% RSLogix 500 project I2P JOB 13 B - Andrew.RSS, saved by version 10.00.00.00 %
PROJECT "ML05B"    % processor: Bul.1763 MicroLogix 1100 Series B %

PROGRAM FILES
  LAD 2   13 rungs

DATA FILES
  O0 OUTPUT  4 elements
  I1 INPUT  6 elements
  S2 STATUS  66 elements
  B3 BINARY  2 elements
  T4 TIMER  1 elements
  C5 COUNTER  1 elements
  R6 CONTROL  1 elements
  N7 INTEGER  1 elements
  F8 FLOAT  1 elements

LADDER 2
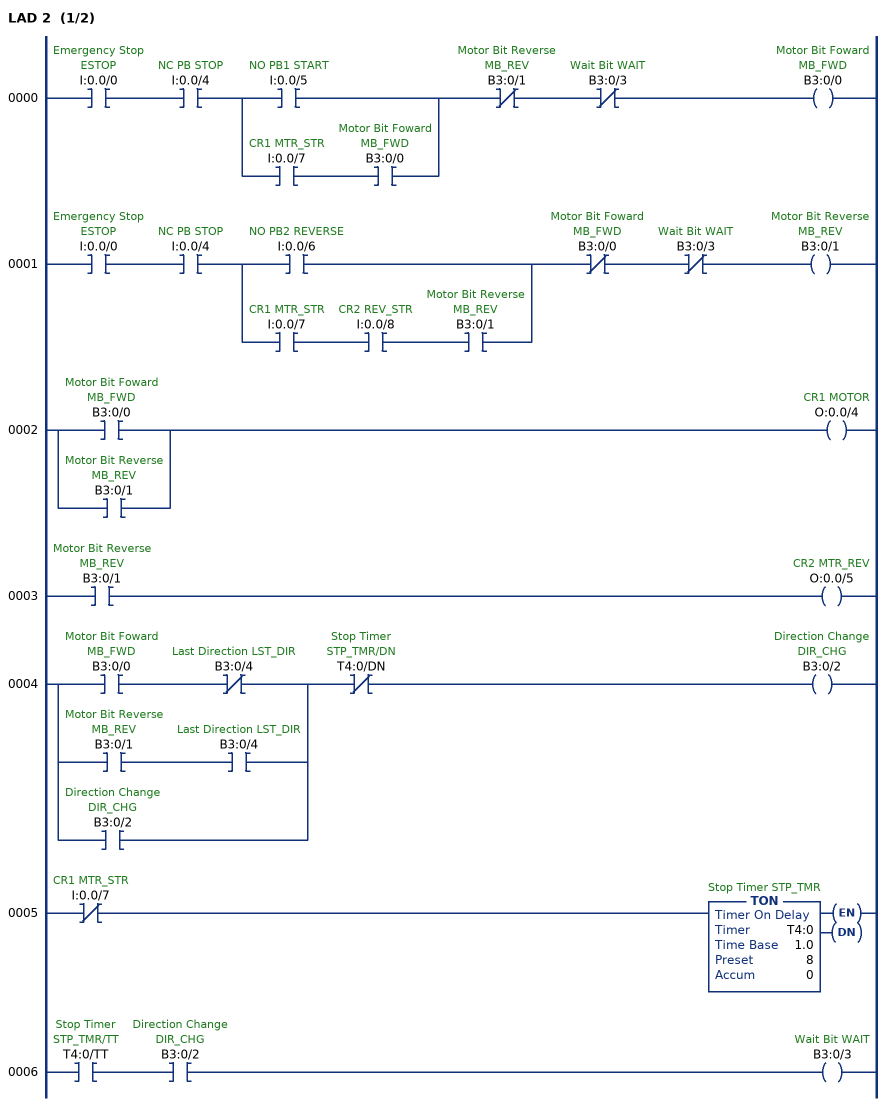
% Rung: 0 %
SOR XIC I:0.0/0 XIC I:0.0/4 BST XIC I:0.0/5 NXB XIC I:0.0/7 XIC B3:0/0 BND XIO B3:0/1 XIO B3:0/3 OTE B3:0/0 EOR
%   I:0.0/0  ESTOP  "Emergency Stop" %
%   I:0.0/4  STOP  "NC PB" %
%   I:0.0/5  START  "NO PB1" %
%   I:0.0/7  MTR_STR  "CR1" %
%   B3:0/0  MB_FWD  "Motor Bit Foward" %
%   B3:0/1  MB_REV  "Motor Bit Reverse" %
%   B3:0/3  WAIT  "Wait Bit" %
% Rung: 1 %
SOR XIC I:0.0/0 XIC I:0.0/4 BST XIC I:0.0/6 NXB XIC I:0.0/7 XIC I:0.0/8 XIC B3:0/1 BND XIO B3:0/0 XIO B3:0/3 OTE B3:0/1 EOR
%   I:0.0/0  ESTOP  "Emergency Stop" %
%   I:0.0/4  STOP  "NC PB" %
%   I:0.0/6  REVERSE  "NO PB2" %
%   I:0.0/7  MTR_STR  "CR1" %
%   I:0.0/8  REV_STR  "CR2" %
%   B3:0/1  MB_REV  "Motor Bit Reverse" %
%   B3:0/0  MB_FWD  "Motor Bit Foward" %
%   B3:0/3  WAIT  "Wait Bit" %
% Rung: 2 %
SOR BST XIC B3:0/0 NXB XIC B3:0/1 BND OTE O:0.0/4 EOR
%   B3:0/0  MB_FWD  "Motor Bit Foward" %
%   B3:0/1  MB_REV  "Motor Bit Reverse" %
%   O:0.0/4  MOTOR  "CR1" %
% Rung: 3 %
SOR XIC B3:0/1 OTE O:0.0/5 EOR
%   B3:0/1  MB_REV  "Motor Bit Reverse" %
%   O:0.0/5  MTR_REV  "CR2" %
% Rung: 4 %
SOR BST XIC B3:0/0 XIO B3:0/4 NXB XIC B3:0/1 XIC B3:0/4 NXB XIC B3:0/2 BND XIO T4:0/DN OTE B3:0/2 EOR
%   B3:0/0  MB_FWD  "Motor Bit Foward" %
%   B3:0/4  LST_DIR  "Last Direction" %
%   B3:0/1  MB_REV  "Motor Bit Reverse" %
%   B3:0/2  DIR_CHG  "Direction Change" %
%   T4:0  STP_TMR  "Stop Timer" %
% Rung: 5 %
SOR XIO I:0.0/7 TON T4:0 1.0 8 0 EOR
%   I:0.0/7  MTR_STR  "CR1" %
%   T4:0  STP_TMR  "Stop Timer" %
% Rung: 6 %
SOR XIC T4:0/TT XIC B3:0/2 OTE B3:0/3 EOR
%   T4:0  STP_TMR  "Stop Timer" %
%   B3:0/2  DIR_CHG  "Direction Change" %
%   B3:0/3  WAIT  "Wait Bit" %

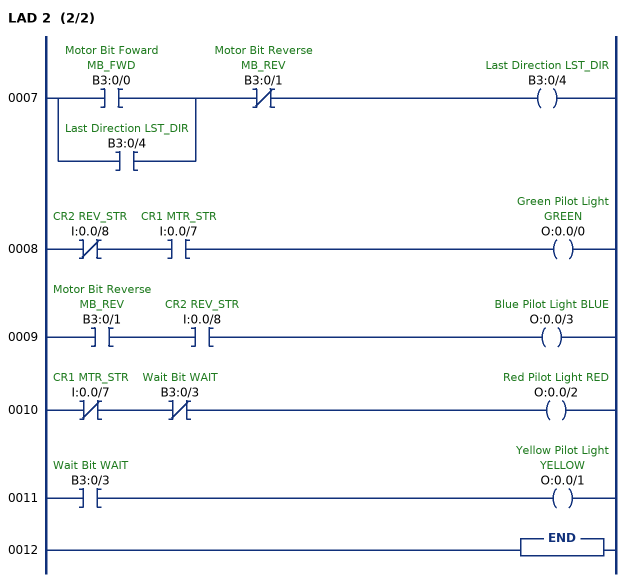
% Rung: 7 %
SOR BST XIC B3:0/0 NXB XIC B3:0/4 BND XIO B3:0/1 OTE B3:0/4 EOR
%   B3:0/0  MB_FWD  "Motor Bit Foward" %
%   B3:0/4  LST_DIR  "Last Direction" %
%   B3:0/1  MB_REV  "Motor Bit Reverse" %
% Rung: 8 %
SOR XIO I:0.0/8 XIC I:0.0/7 OTE O:0.0/0 EOR
%   I:0.0/8  REV_STR  "CR2" %
%   I:0.0/7  MTR_STR  "CR1" %
%   O:0.0/0  GREEN  "Green Pilot Light" %
% Rung: 9 %
SOR XIC B3:0/1 XIC I:0.0/8 OTE O:0.0/3 EOR
%   B3:0/1  MB_REV  "Motor Bit Reverse" %
%   I:0.0/8  REV_STR  "CR2" %
%   O:0.0/3  BLUE  "Blue Pilot Light" %
% Rung: 10 %
SOR XIO I:0.0/7 XIO B3:0/3 OTE O:0.0/2 EOR
%   I:0.0/7  MTR_STR  "CR1" %
%   B3:0/3  WAIT  "Wait Bit" %
%   O:0.0/2  RED  "Red Pilot Light" %
% Rung: 11 %
SOR XIC B3:0/3 OTE O:0.0/1 EOR
%   B3:0/3  WAIT  "Wait Bit" %
%   O:0.0/1  YELLOW  "Yellow Pilot Light" %
% Rung: 12 %
SOR END EOR

OTHER DOCUMENTED ADDRESSES
  AI  
  B3:1  BIT2  "Bit2"
  I:0.0/1  FWD  "3 Position Selector Switch, A"
  I:0.0/2  REV  "3 Position Selector Switch, B"
  I:0.0/3  JOG_RUN  "2 Position Selector Switch"
  NC_PB  "NC PB"

DATA TABLE (non-zero values as saved)
DATA T4
% .PRE .ACC %
% T4:0 % 8 0
